// TIA Portal V17 export
// export: Created 2024-10-17T14:16:15.8752117Z, ExportSetting WithDefaults, DisplayName Totally Integrated Automation Portal, DisplayVersion V17 Update 4, DisplayName TIA Portal Openness, DisplayVersion V17 Update 4, DisplayName TIA Portal Version Control Interface, DisplayVersion V17, DisplayName SINAMICS Startdrive Advanced, DisplayVersion V17 Update2, DisplayName SINAMICS Startdrive G130, G150, S120, S150, SINAMICS MV, S210, DisplayVersion V17 Update2, DisplayName SINAMICS Startdrive G110M, G120, G120C, G120D, G120P, G115D, DisplayVersion V17 Update2, DisplayName STEP 7 Professional, DisplayVersion V17 Update 4, DisplayName STEP 7 Safety, DisplayVersion V17, DisplayName WinCC Advanced / Unified PC, DisplayVersion V17 Update 4
DATA_BLOCK "UnitModeStateManagerDiagnosticsForHMI"   // DB30134
{ S7_Optimized_Access := 'TRUE'; DB_Accessible_From_OPC_UA := 'FALSE' }
VERSION : 0.1
// stored: AutoNumber true, DBAccessibleFromOPCUA false, DBAccessibleFromWebserver false, IsOnlyStoredInLoadMemory false, IsRetainMemResEnabled false, IsWriteProtectedInAS false, MemoryReserve 0
   VAR
      actualDiagnosticsBufferIndex { ExternalWritable := 'False'} : Int;   // Index of the actual diagnostics buffer entry of the LPMLV2022_UnitModeStateManager (InstLPMLV2022_UnitModeStateManager.diagnostics.bufferIndex)
      diagnosticsBufferIndexForHMI : Int;   // Index for selecting the diagnostics buffer entry to be displayed on the HMI
      diagnosticsBufferEntryForHMI { ExternalWritable := 'False'} : "LPMLV2022_typeDiagnosticsEntry";   // Selected diagnostics buffer entry (InstLPMLV2022_UnitModeStateManager.diagnostics.buffer[diagnosticsBufferIndexForHMI])
      messageCurrentPLCIndex { ExternalWritable := 'False'} : Byte;   // Message of the actual diagnostics buffer entry of the LPMLV2022_UnitModeStateManager
   END_VAR
BEGIN
END_DATA_BLOCK
